PROGRAM MAIN
VAR
	Influx : To_InfluxDb;
	bExecute: BOOL;
	tTime: TIME := T#1s;
	bBusy: BOOL;
	bError: BOOL;
	bErrorId: DINT;
	stSensors : ARRAY[0..10] OF ST_SensorData;
	Generatedata : FBGenerateData;
	tIntervalTimer: TON;
	sHostName: STRING;
END_VAR

stSensors[0].sSensorId := '1PT01';
Generatedata(data:=stSensors[0]);
stSensors[1].sSensorId := '1PT02';
Generatedata(data:=stSensors[1]);
stSensors[2].sSensorId := '1PT03';
Generatedata(data:=stSensors[2]);
stSensors[3].sSensorId := '1PT04';
Generatedata(data:=stSensors[3]);
stSensors[4].sSensorId := '1PT05';
Generatedata(data:=stSensors[4]);
stSensors[5].sSensorId := '1PT06';
Generatedata(data:=stSensors[5]);


// Send data to InfluxDb
Influx(
	bExecute:= bExecute, 
	tInterval:= tTime, 
	sHostName:= '127.0.0.1', 
	nHostPort:= 8086, 
	sDatabaseName:= 'SensorData',
	sMeasurementName:= 'PtData',
	stData:= stSensors, 
	bBusy=> bBusy, 
	bError=> bError, 
	nErrId=> bErrorId);

END_PROGRAM

(* stored: Version 1.1.0.1, ProductVersion 3.1.4024.9
   POU MAIN: Id {709da0b2-f321-4915-b743-e457665273bf}, SpecialFunc None *)
